INTERFACE I_ResultFile EXTENDS __SYSTEM.IQueryInterface

METHOD AddTestCaseResult
VAR_INPUT
END_VAR
END_METHOD

METHOD AddTestSuite
VAR_INPUT
END_VAR
END_METHOD

METHOD Initialize
VAR_INPUT
END_VAR
END_METHOD

METHOD Save
VAR_INPUT
END_VAR
END_METHOD

END_INTERFACE

(* stored: Version 1.1.0.1
   Itf I_ResultFile: Id {e1366dc8-517e-46ad-b1e3-80eafaf62fca}
   Method AddTestCaseResult: Id {3b1e675c-601a-4597-82c3-21011f29cf49}
   Method AddTestSuite: Id {336643ed-f4f2-4062-ab5f-cbc7284ffffe}
   Method Initialize: Id {7c254bb1-9728-4958-adfe-eece97237b3f}
   Method Save: Id {690c3506-9c68-4a55-8088-e8b719c43680} *)
